Staubli VAL3: feedbackStatus.pgx

public program feedbackStatus(num x_nOutConnFlag)
begin

  // update connection status on port 11002 (feedback server)

  gotoxy(scMonitor, 0,3)
  // 11 characters: gotoxy(12,3) to insert status
  put(scMonitor, "Port 11002:")
  gotoxy(scMonitor, 12,3)
  switch x_nOutConnFlag
    case -1
      put(scMonitor, "connection lost")
    break
    case 0
      put(scMonitor, "not connected")
    break
    case 1
      put(scMonitor, "connected")
    break
    default
      put(scMonitor, "not connected")
    break
  endSwitch

end
